// TIA Portal project "TOF ile Zamanlayıcı Uygulaması_2" (V18)

(* hardware
DEVICE "S7-1200 station_1"  S7-1200 Station
   slot 0: "Rack_0"  S7-1200 Rack  Rack  V1.0
   slot 1: "PLC_1"  CPU 1214C AC/DC/Rly  6ES7 214-1BG40-0XB0  V4.6
*)

// ===== PLC "PLC_1"  CPU 1214C AC/DC/Rly =====

VAR_GLOBAL   // PLC tag table "Default tag table"
   "Stop" AT %I0.0 : Bool;
   "Start" AT %I0.1 : Bool;
   "Motor_1" AT %Q0.0 : Bool;
   "Tag_1" AT %M0.0 : Bool;
END_VAR

// folder: System blocks/Program resources

DATA_BLOCK "IEC_Timer_0_DB_1"   // DB1
{ S7_Optimized_Access := 'TRUE' }
AUTHOR : Simatic
FAMILY : IEC
NAME : IEC_TMR
VERSION : 1.0
// stored: InstanceOfName IEC_TIMER
"IEC_TIMER"
BEGIN
END_DATA_BLOCK

DATA_BLOCK "IEC_Timer_0_DB"   // DB2
{ S7_Optimized_Access := 'TRUE' }
AUTHOR : Simatic
FAMILY : IEC
NAME : IEC_TMR
VERSION : 1.0
// stored: InstanceOfName IEC_TIMER
"IEC_TIMER"
BEGIN
END_DATA_BLOCK

// folder: (top level)

ORGANIZATION_BLOCK "Main"   // OB1, LAD, ProgramCycle
TITLE = "Main Program Sweep (Cycle)"
{ S7_Optimized_Access := 'TRUE' }
VERSION : 0.1
// Start butonuna basıldığında motorumuz hemen çalışmaya başlayacak.
// 20sn sonra motor kendisi duracaktır.
   VAR_INPUT
      Initial_Call : Bool;   // Initial call of this OB
      Remanence : Bool;   // =True, if remanent data are available
   END_VAR
BEGIN

REGION Network 1
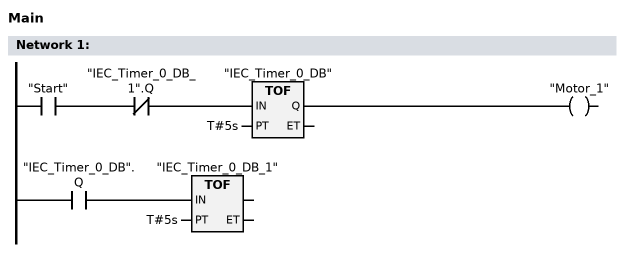
   "IEC_Timer_0_DB".TOF(IN := "Start" AND NOT "IEC_Timer_0_DB_1".Q, PT := T#5s);
   "Motor_1" := "IEC_Timer_0_DB".Q;
   "IEC_Timer_0_DB_1".TOF(IN := "IEC_Timer_0_DB".Q, PT := T#5s);
END_REGION
END_ORGANIZATION_BLOCK